TYPE ST_DefinitionDO :
STRUCT
	Name						: STRING := '';
	Description					: STRING := '';
END_STRUCT
END_TYPE

(* stored: Version 1.1.0.1, ProductVersion 3.1.4026.18
   DUT ST_DefinitionDO: Id {36d4a399-76fd-462c-881a-a2554247b29e} *)
